PROGRAM PRG_TestSimpleApi
VAR
	bExecute		: BOOL;
	bExecuteSingle	: BOOL;
	
	nArg			: INT := 42;
	sArg			: T_MaxString := 'foo';
	fArg			: REAL := 4.2;
END_VAR

IF bExecute OR bExecuteSingle THEN
	bExecuteSingle := FALSE;
	
	F_LogLA3(
		E_LogLevel.eInfo,
		'PRG_TestSimpleApi',
		'Log F_LogLA3({arg1},{arg2},{arg3})',
		nArg,
		sArg,
		fArg
	);
	
	F_LogA3(
		E_LogLevel.eInfo,
		'Log F_LogA3({arg1},{arg2},{arg3})',
		nArg,
		sArg,
		fArg
	);
	
END_IF

END_PROGRAM

(* stored: Version 1.1.0.1, ProductVersion 3.1.4024.0
   POU PRG_TestSimpleApi: Id {bcc7908d-3a35-4ae4-afd2-9b6ede60025b}, SpecialFunc None *)
